// TIA Portal V17 export
// export: Created 2023-05-07T12:12:21.8991322Z, ExportSetting WithDefaults, DisplayName Totally Integrated Automation Portal, DisplayVersion V17, DisplayName TIA Portal Openness, DisplayVersion V17, DisplayName TIA Portal Version Control Interface, DisplayVersion V17, DisplayName TIA Portal Test Suite Advanced, DisplayVersion V17, DisplayName STEP 7 Professional, DisplayVersion V17, DisplayName SIMATIC Energy Suite, DisplayVersion V17, DisplayName STEP 7 Safety, DisplayVersion V17, DisplayName WinCC Professional, DisplayVersion V17
FUNCTION "ShowPompOn" : Void   // FC6, LAD
TITLE = ShowPompOn
{ S7_Optimized_Access := 'TRUE' }
VERSION : 0.1
// stored: AutoNumber true, IsIECCheckEnabled false, SetENOAutomatically false, UDAEnableTagReadback false
   VAR_TEMP   // added for the SCL form of the ladder/FBD networks
      _w1 : Bool;
   END_VAR
BEGIN

REGION Network 1: Move: TopPump
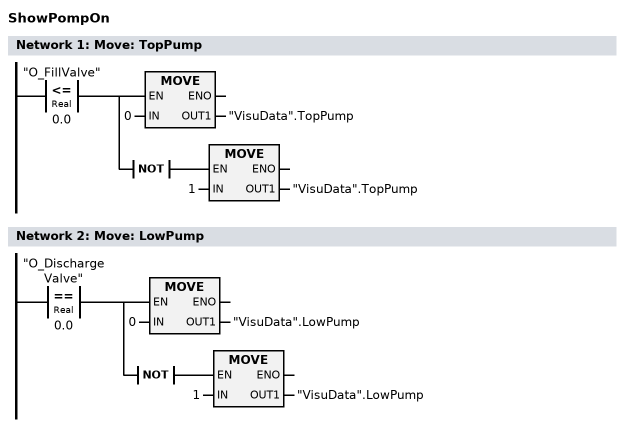
   RUNG wire#powerrail
      { S7_Templates := "SrcType := Real" } LE_Contact(in1 := "O_FillValve", in2 := 0.0)
      wire#w1
      Move(in := 0, out1 => "VisuData".TopPump)
   END_RUNG
   RUNG wire#w1
      Not()
      Move(in := 1, out1 => "VisuData".TopPump)
   END_RUNG
   // the same network as SCL:
   #_w1 := "O_FillValve" <= 0.0;
   IF #_w1 THEN "VisuData".TopPump := 0; END_IF;
   IF NOT #_w1 THEN "VisuData".TopPump := 1; END_IF;
END_REGION

REGION Network 2: Move: LowPump
   RUNG wire#powerrail
      { S7_Templates := "SrcType := Real" } EQ_Contact(in1 := "O_DischargeValve", in2 := 0.0)
      wire#w1
      Move(in := 0, out1 => "VisuData".LowPump)
   END_RUNG
   RUNG wire#w1
      Not()
      Move(in := 1, out1 => "VisuData".LowPump)
   END_RUNG
   // the same network as SCL:
   #_w1 := "O_DischargeValve" = 0.0;
   IF #_w1 THEN "VisuData".LowPump := 0; END_IF;
   IF NOT #_w1 THEN "VisuData".LowPump := 1; END_IF;
END_REGION
END_FUNCTION
